PROGRAM F_DUCHAS
VAR_INPUT
	Func:E_funcio;
	
END_VAR
VAR
	///Activa
	xActv: BOOL;
	///Fin Funcion
	xFiFunc: BOOL;
	
	tFinDuchas: Ton;
	Z_Spray: BOOL;
END_VAR


(*Activa funcio *)
xActv:= func.Actv_Funcio;

(*FIN FUNCION*)
		xFiFunc				:=	xActv AND 
							NOT (
							F_FIN_DUCHAS.xActv OR
							F_VACIADO.xActv
							);

(*ACTIVA SALIDAS*)
Z_Spray:=xActv ;

END_PROGRAM

(* stored: Version 1.1.0.1, ProductVersion 3.1.4024.10
   POU F_DUCHAS: Id {16155bfb-b06d-4868-a8a1-af0c864abf0e}, SpecialFunc None *)
